# B&R Automation Studio project lab2-Control-software-for-mech-safe-door-control-module
Automation Studio 4.5.2.102

## Configuration SampleText

### Hardware
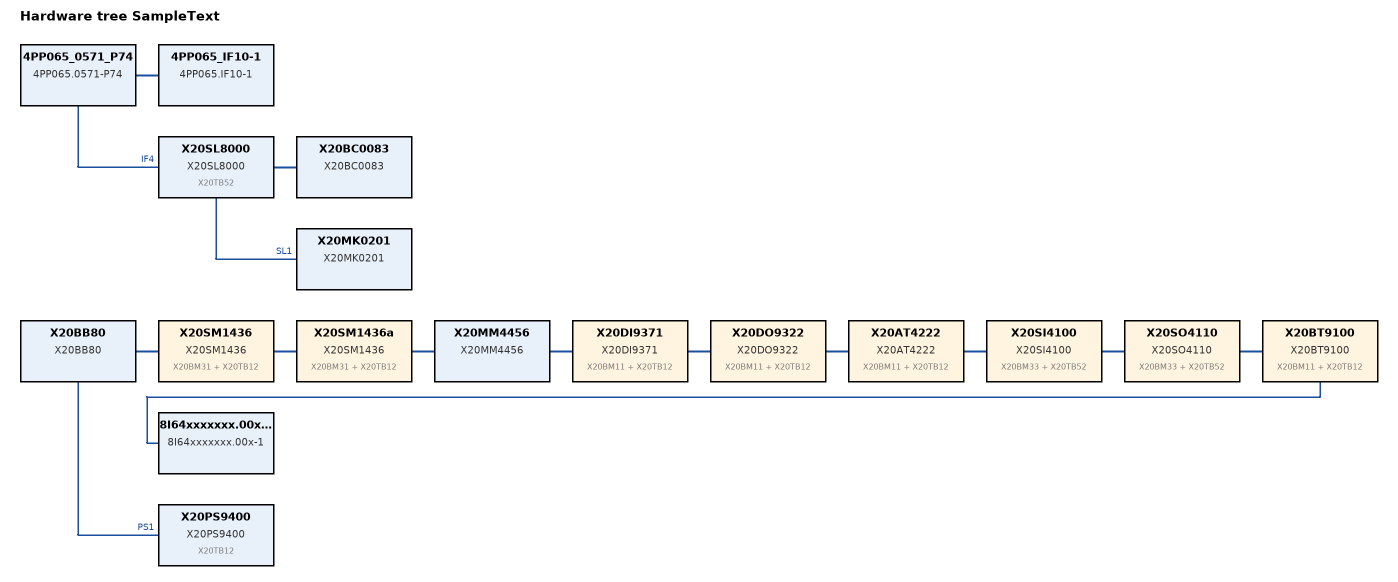
```
4PP065_0571_P74 : 4PP065.0571-P74 v1.1.2.0
  Connector IF5:
    ActivateDevice = 1
    Mode = Manual
    InternetAddress = 10.0.1.13
    SubnetMask = 255.255.255.0
  ConfigurationID = labBR
  TimerDeviceType = EPLX2X
  TimerDevice = 4PP065_0571_P74.IF4
  TaskClassIdleTime = 2000
  Cyclic1Duration = 2000
  Cyclic1Tolerance = 0
  Cyclic1Output = 1
4PP065_IF10-1 : 4PP065.IF10-1 v1.0.3.0  [SS -> 4PP065_0571_P74.SS1]
8I64xxxxxxx.00x-1 : 8I64xxxxxxx.00x-1 v1.3.9.1  [X2X1 -> X20BT9100.X2X1 [Cable Type=X2XCable, Length=10, Version=1.0.0.2]]
  FunctionModel = Standard
  packedETAD = packed
  packedETI = packed
  packedCMDD = packed
  packedCMI = packed
X20AT4222 : X20AT4222 v1.2.3.0  [SS1 -> X20TB12e.SS; SL -> X20BM11c.SL1]
X20BB80 : X20BB80 v1.0.2.0
X20BC0083 : X20BC0083 v2.7.0.0  [PLK1 -> X20SL8000.PLK2 (NodeNumber=2) [Cable Type=PowerlinkCable, Length=10, Version=1.0.0.2]; SL -> X20BB80.SL1]
X20BM11 : X20BM11 v1.0.0.1  [X2X1 -> X20BM33a.X2X2]
X20BM11a : X20BM11 v1.0.0.1  [X2X1 -> X20MM4456.X2X2]
X20BM11b : X20BM11 v1.0.0.1  [X2X1 -> X20BM11a.X2X2]
X20BM11c : X20BM11 v1.0.0.1  [X2X1 -> X20BM11b.X2X2]
X20BM31 : X20BM31 v1.0.0.1  [X2X1 -> X20BB80.IF1]
X20BM31a : X20BM31 v1.0.0.1  [X2X1 -> X20BM31.X2X2]
X20BM33 : X20BM33 v1.0.0.4  [X2X1 -> X20BM11c.X2X2]
X20BM33a : X20BM33 v1.0.0.4  [X2X1 -> X20BM33.X2X2]
X20BT9100 : X20BT9100 v1.0.3.0  [SS1 -> X20TB12f.SS; SL -> X20BM11.SL1]
X20DI9371 : X20DI9371 v1.0.2.0  [SS1 -> X20TB12c.SS; SL -> X20BM11a.SL1]
X20DO9322 : X20DO9322 v1.0.3.0  [SS1 -> X20TB12d.SS; SL -> X20BM11b.SL1]
X20MK0201 : X20MK0201 v1.0.0.0  [SL -> X20SL8000.SL1]
X20MM4456 : X20MM4456 v1.1.5.0  [X2X1 -> X20BM31a.X2X2]
X20PS9400 : X20PS9400 v1.0.2.4  [SS1 -> X20TB12.SS; PS -> X20BB80.PS1]
X20SI4100 : X20SI4100 v1.10.1.1  [SS1 -> X20TB52.SS; SL -> X20BM33.SL1]
X20SL8000 : X20SL8000 v1.6.5.1  [PLK1 -> 4PP065_0571_P74.IF4 (NodeNumber=1) [Cable Type=PowerlinkCable, Length=10, Version=1.0.0.2]; PLK2 -> X20BC0083.PLK1 (NodeNumber=1) [Cable Type=PowerlinkCable, Length=10, Version=1.0.0.2]; SS1 -> X20TB52b.SS]
  SafeProject = SafeLOGIC-1
X20SM1436 : X20SM1436 v1.4.2.1  [SS1 -> X20TB12a.SS; SL -> X20BM31.SL1]
X20SM1436a : X20SM1436 v1.4.2.1  [SS1 -> X20TB12b.SS; SL -> X20BM31a.SL1]
X20SO4110 : X20SO4110 v1.10.1.1  [SS1 -> X20TB52a.SS; SL -> X20BM33a.SL1]
  SafeModuleID = 3
X20TB12 : X20TB12 v1.0.0.0
X20TB12a : X20TB12 v1.0.0.0
X20TB12b : X20TB12 v1.0.0.0
X20TB12c : X20TB12 v1.0.0.0
X20TB12d : X20TB12 v1.0.0.0
X20TB12e : X20TB12 v1.0.0.0
X20TB12f : X20TB12 v1.0.0.0
X20TB52 : X20TB52 v1.0.0.1
X20TB52a : X20TB52 v1.0.0.1
X20TB52b : X20TB52 v1.0.0.1
```

## Logical view

### Global.var
```iecst
VAR
	gAxis01 : ACP10AXIS_typ := (0);
	gAxis01_HW : SdcHwCfg_typ := (0);
	gAxis01_DrvIf : SdcDrvIf16_typ := (0);
	gAxis01_DiDoIf : SdcDiDoIf_typ := (0);
	gAxis01_ModuleOk : BOOL := 0;
END_VAR
```
